PROGRAM Device_POU
VAR
	fbCylinderBase:ARRAY [0..20] OF  FB_CylinderBase;
END_VAR


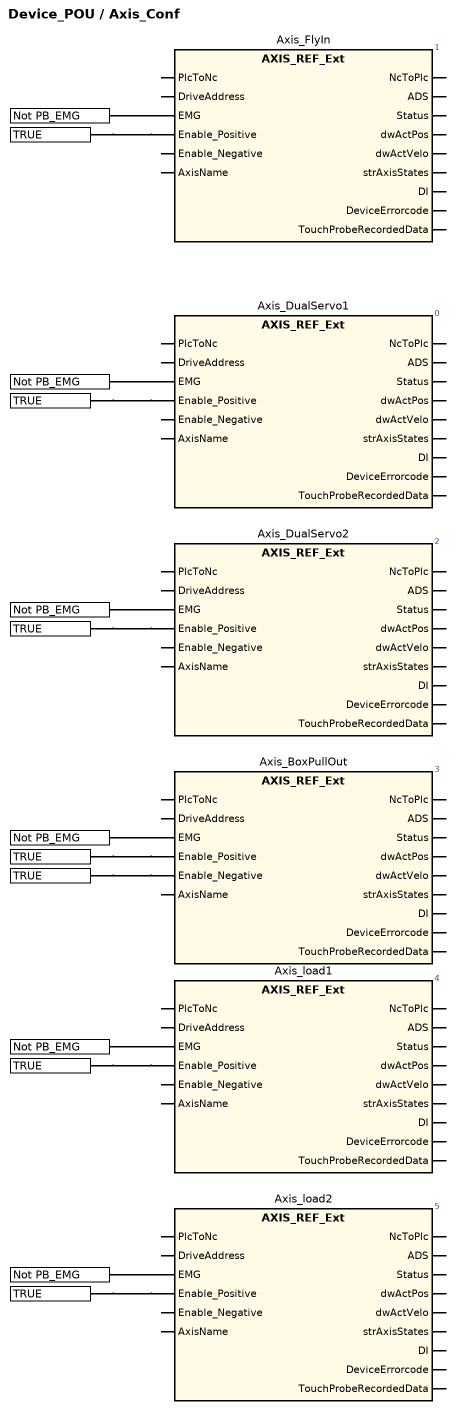
// PAGE Axis_Conf
Axis_DualServo1(EMG := Not PB_EMG, Enable_Positive := TRUE); // AXIS_REF_Ext
Axis_FlyIn(EMG := Not PB_EMG, Enable_Positive := TRUE); // AXIS_REF_Ext
Axis_DualServo2(EMG := Not PB_EMG, Enable_Positive := TRUE); // AXIS_REF_Ext
Axis_BoxPullOut(EMG := Not PB_EMG, Enable_Positive := TRUE, Enable_Negative := TRUE); // AXIS_REF_Ext
Axis_load1(EMG := Not PB_EMG, Enable_Positive := TRUE); // AXIS_REF_Ext
Axis_load2(EMG := Not PB_EMG, Enable_Positive := TRUE); // AXIS_REF_Ext

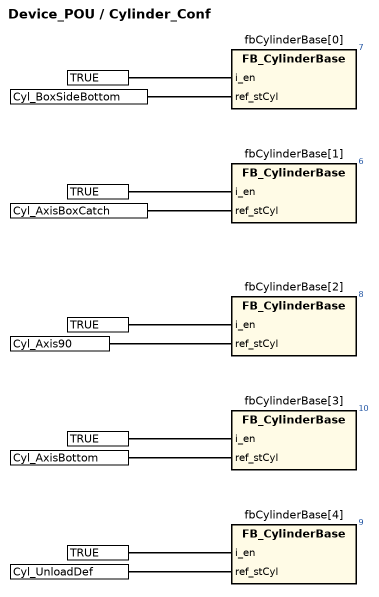
// PAGE Cylinder_Conf
fbCylinderBase[1](i_en := TRUE, ref_stCyl := Cyl_AxisBoxCatch); // FB_CylinderBase
fbCylinderBase[0](i_en := TRUE, ref_stCyl := Cyl_BoxSideBottom); // FB_CylinderBase
fbCylinderBase[2](i_en := TRUE, ref_stCyl := Cyl_Axis90); // FB_CylinderBase
fbCylinderBase[4](i_en := TRUE, ref_stCyl := Cyl_UnloadDef); // FB_CylinderBase
fbCylinderBase[3](i_en := TRUE, ref_stCyl := Cyl_AxisBottom); // FB_CylinderBase

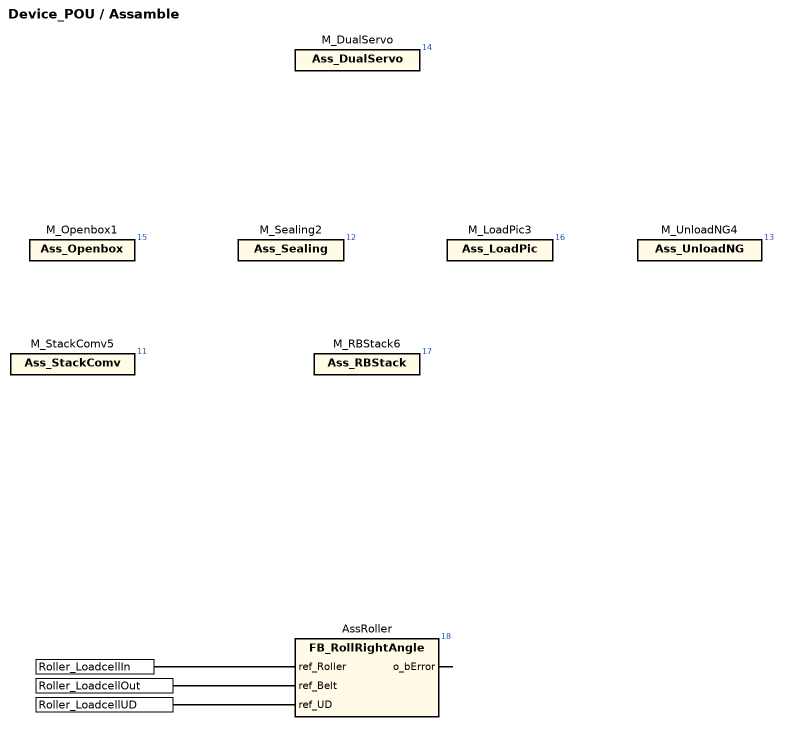
// PAGE Assamble
M_StackComv5(); // Ass_StackComv
M_Sealing2(); // Ass_Sealing
M_UnloadNG4(); // Ass_UnloadNG
M_DualServo(); // Ass_DualServo
M_Openbox1(); // Ass_Openbox
M_LoadPic3(); // Ass_LoadPic
M_RBStack6(); // Ass_RBStack
AssRoller(ref_Roller := Roller_LoadcellIn, ref_Belt := Roller_LoadcellOut, ref_UD := Roller_LoadcellUD); // FB_RollRightAngle

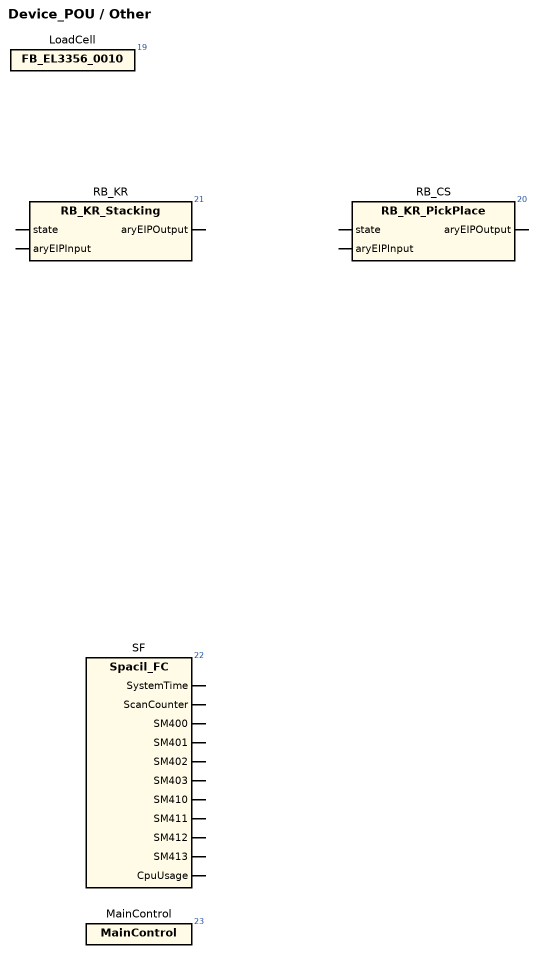
// PAGE Other
LoadCell(); // FB_EL3356_0010
RB_CS(); // RB_KR_PickPlace
RB_KR(); // RB_KR_Stacking
SF(); // Spacil_FC
MainControl();

END_PROGRAM

(* stored: Version 1.1.0.1, ProductVersion 3.1.4026.18
   POU Device_POU: Id {892213d6-fbc5-482a-b840-a0aa33a71c3e}, SpecialFunc None *)
